FUNCTION_BLOCK TestModule_3
VAR_INPUT
	fbNextStationReleaseHybrid : ReleaseHybrid;
END_VAR
VAR_OUTPUT
END_VAR
VAR
END_VAR

fbNextStationReleaseHybrid();

END_FUNCTION_BLOCK

(* stored: Version 1.1.0.1, ProductVersion 3.1.4024.2
   POU TestModule_3: Id {80aeded2-fde7-42a7-be9c-6fe0efe40b0a}, SpecialFunc None *)
